FUNCTION_BLOCK FB_WiezaSygnalizacyjna_Cyfrowe IMPLEMENTS ITF_WiezaSygnalizacyjna
VAR
	bCzerwony						AT%Q*	: BOOL;
	bZolty							AT%Q*	: BOOL;
	bZielony						AT%Q*	: BOOL;
	bNiebieski						AT%Q*	: BOOL;
	bBialy							AT%Q*	: BOOL;
	
END_VAR

(*==================================================================================================
								RJM Maszyny sp. z o.o.
									22.06.2022
	Wlaczanie/Wylaczenia segment bialy   
 	v1.0	|| TC v 3.1.4024.29		|| - pierwsza wersja
==================================================================================================*)
PROPERTY Bialy : BOOL
GET
Bialy										:= bBialy;
END_GET
SET
bBialy										:= Bialy;
END_SET
END_PROPERTY

(*==================================================================================================
								RJM Maszyny sp. z o.o.
									22.06.2022
	Wlaczanie/Wylaczenia segment czerwony   
 	v1.0	|| TC v 3.1.4024.29		|| - pierwsza wersja
==================================================================================================*)
PROPERTY Czerwony : BOOL
GET
Czerwony									:= bCzerwony;
END_GET
SET
bCzerwony									:= Czerwony;
END_SET
END_PROPERTY

(*==================================================================================================
								RJM Maszyny sp. z o.o.
									22.06.2022
	Wlaczanie/Wylaczenia segment niebieski   
 	v1.0	|| TC v 3.1.4024.29		|| - pierwsza wersja
==================================================================================================*)
PROPERTY Niebieski : BOOL
GET
Niebieski									:= bNiebieski;
END_GET
SET
bNiebieski									:= Niebieski;
END_SET
END_PROPERTY

(*==================================================================================================
								RJM Maszyny sp. z o.o.
									22.06.2022
	Wlaczanie/Wylaczenia segment zielony  
 	v1.0	|| TC v 3.1.4024.29		|| - pierwsza wersja
==================================================================================================*)
PROPERTY Zielony : BOOL
GET
Zielony										:= bZielony;
END_GET
SET
bZielony									:= Zielony;
END_SET
END_PROPERTY

(*==================================================================================================
								RJM Maszyny sp. z o.o.
									22.06.2022
	Wlaczanie/Wylaczenia segment zolty   
 	v1.0	|| TC v 3.1.4024.29		|| - pierwsza wersja
==================================================================================================*)
PROPERTY Zolty : BOOL
GET
Zolty										:= bZolty;
END_GET
SET
bZolty										:= Zolty;
END_SET
END_PROPERTY

END_FUNCTION_BLOCK

(* stored: Version 1.1.0.1, ProductVersion 3.1.4024.11
   POU FB_WiezaSygnalizacyjna_Cyfrowe: Id {3a8c2e0e-0d8b-4d99-aca2-93bac4cc37df}, SpecialFunc None
   Property Bialy: Id {f4b7929b-5bb9-4c08-9e35-c2e6090d98e7}
   Get Get: Id {a97d4511-e3db-406e-823b-bf829057ecc1}
   Set Set: Id {03e4a57e-21e5-4f60-8e98-70494430c300}
   Property Czerwony: Id {bf1972cd-37a2-4362-93bb-07214392fb65}
   Get Get: Id {57eefb78-838a-4f5f-a261-261198c249ef}
   Set Set: Id {c5011a76-a9dc-4a6c-bb19-1142af4e22d0}
   Property Niebieski: Id {4d8cffb8-e1c8-4696-bac4-6476a4944a69}
   Get Get: Id {b55a68f0-e5e3-4257-bd94-18bbecd83250}
   Set Set: Id {5ca4def4-ddfe-4c66-9ff6-850020d0343f}
   Property Zielony: Id {b0bf2c0f-1b9b-4ae4-99c2-b2afd64cb06d}
   Get Get: Id {abeb282b-6e43-4ad3-8470-8d6ddc6f4e40}
   Set Set: Id {675701ae-0ab2-4957-a980-32260458028f}
   Property Zolty: Id {1b747b60-9574-460f-a783-f6f2fdd7fb73}
   Get Get: Id {057ecf5f-1452-4ee3-99c3-3793618016ef}
   Set Set: Id {350806d8-06b8-4fa6-b44b-5291f7be0217} *)
